{attribute addProperty BoxType "EL2622-0010-0016"}
{attribute addProperty Id "InputsAT %I*Inputs_BDF19946810ChannelAT %Q*ARRAY[0..1] OF Channel_7F374EB01620WcStateAT %I*WcState_F855686C1620InfoDataAT %I*InfoData_192954DE1620"}
{attribute addProperty CRC "772639126"}
{attribute addProperty SizeInBites "56"}
{attribute addProperty SizeInBytes "7"}
TYPE EL2622_0939F1F7 :
STRUCT
	{attribute addProperty Name "Inputs"}
	Inputs : Inputs_BDF19946;
	{attribute addProperty Name "Channel"}
	Channel : ARRAY[0..1] OF Channel_7F374EB0;
	{attribute addProperty Name "WcState"}
	WcState : WcState_F855686C;
	{attribute addProperty Name "InfoData"}
	InfoData : InfoData_192954DE;
END_STRUCT
END_TYPE

(* stored: Version 1.2.0.0, ProductVersion 3.1.4024.9
   DUT EL2622_0939F1F7: Id {dc754e69-7fba-42b0-8337-8d9092b28d09} *)
